// Struct contains all data from other tasks and controller used for master control
TYPE ST_MasterInputDataPool :
STRUCT
		
	// UI information, import from UI controller
	m_UIData AT %I*:ST_UIData;
	
	// safety information, import from safety check task
	m_safetyData AT %I*: ST_CartStatus;
	
	// cart information, import from other task
	m_cartStatus AT %I*:ST_CartStatus;
	
	// slave robot information, import from other device
	m_slaveStatus AT %I*:ST_SlaveStatus;
	
END_STRUCT
END_TYPE

(* stored: Version 1.1.0.1, ProductVersion 3.1.4024.12
   DUT ST_MasterInputDataPool: Id {8edc6f5a-e934-4abf-9384-df71872be806} *)
